PROGRAM MAIN
VAR
	SoftClock : RTC_EX;
	Chirp :fb_chirpgen;
	outputval: LREAL;
END_VAR

.Global_Variables.TcJoy(); // Read HMI data
 // read drive limit input swtich status
 io.Drive1positivelimitSw := io.Drive1digitalinBtyes[2].4;
 io.Drive1NegativelimitSw := io.Drive1digitalinBtyes[2].5;
 io.Drive2positivelimitSw := io.Drive2digitalinBtyes[2].4;
 io.Drive2NegativelimitSw := io.Drive2digitalinBtyes[2].5;
P_HMI_polling();
IF .Global_Variables.TcJoy.bIsActive THEN // if HMI is connected
	;
END_IF
p_singenerator();

chirp(en := TRUE, Reset :=FALSE, Offset := 10.0, A := 15, w1 := 10, w2 := 25,M :=2000, SignalOut => outputval);


p_FaultMonitoring(); // Check fault routine
//inputs
p_TextModeRead();
//Seq
//Outputs
P_FunctionGenerators();

SoftClock(En := Global_Variables.EnablemsClock,PMSEK:=0, Q=> Global_Variables.msClockValid);// Call for a 1ms resolution software timer to start at 0ms when enable goes true.
p_MotorControl_ST();
p_MotorControl();

//logging
//recipe system

END_PROGRAM

(* stored: Version 1.1.0.1, ProductVersion 3.1.4024.4
   POU MAIN: Id {d25881fd-bae0-4e0a-b3eb-c173027ef094}, SpecialFunc None *)
